FUNCTION_BLOCK FB_DC
VAR_INPUT
END_VAR
VAR_OUTPUT
	bStatusOn : BOOL;
END_VAR
VAR
	OPC_UA				: FB_OPC_UA_READ;
	stOPC_UA_Server		: ST_OPC_UA_Server;
	sOPC_UA_Server_URL 	: STRING;
	sNamespaceName		: STRING;
	aNodes				: ARRAY[1..1] OF ST_OPC_UANode;
	nNodeCount			: UDINT := 1;
	stIndexRange		: ARRAY [1..nMaxIndexRange] OF ST_UAIndexRange;
	currentNode			: UDINT := 1;
	
	bStatusOn_CoolingLubricant : BOOL;
	bStatusOn_Machine : BOOL;
END_VAR

sOPC_UA_Server_URL 	:= GlobalVariables.sIP_DC;
sNamespaceName 		:= 'http://www.boschrexroth.com/IndraLogic';

(*Define Nodes to Read*)
aNodes[1].NodeID.sIdentifier			:= '.bHMU_DCBusCharged';
aNodes[1].NodeID.eIdentifierType		:= eUAIdentifierType_String;
aNodes[1].SizeOfDataType				:= DINT_TO_UDINT(eUAType_Boolean);
aNodes[1].NodeAddInfo.nIndexRangeCount 	:= 0;
aNodes[1].NodeAddInfo.stIndexRange		:= stIndexRange;
aNodes[1].TargetVar						:= ADR(bStatusOn);

OPC_UA(
	stNode				:= aNodes[currentNode],
	sOPC_UA_Server_Url 	:= sOPC_UA_Server_URL,
	sNamespaceName		:= sNamespaceName);
currentNode := currentNode + 1;
IF currentNode > nNodeCount THEN
	currentNode := 1;
END_IF

END_FUNCTION_BLOCK

(* stored: Version 1.1.0.1, ProductVersion 3.1.4024.10
   POU FB_DC: Id {eaa9fb1e-ba41-4ba1-9971-267c969dd365}, SpecialFunc None *)
